PROGRAM Y_Master_Y_Axis
VAR
	
	// Link to Task
	refY_Axis							:AXIS_REF;	//Axis_1
										
										
	fPositionLimitMin					:LREAL			 := 5;
	fPositionLimitMax					:LREAL			 := 110;
	fLimitPositionLow					:LREAL; 		//16#0001_000D
	fLimitPositionHigh					:LREAL;			//16#0001_000E
	
	// Local Axis Config
	posTarget							:LREAL;
	fOffsets							:ARRAY [1..3]OF LREAL;
	nOfSetPos							:INT:=3;
	fCurrentPosition					:LREAL;

    // State Machine CTRL
    eState								:E_AxisState:=E_AxisState.ABORTED;

	// Timers && Triggers
	tonResetError						:Tc2_Standard.TON;
	tonPowerAxis						:Tc2_Standard.TON;
	tonPowerAxis2						:Tc2_Standard.TON;
	tonActionDone						:Tc2_Standard.TON;
	tonMoveTimeout						:Tc2_Standard.TON;
	tonPowerUpTimeout					:Tc2_Standard.TON;
	tonPowerUpError						:Tc2_Standard.TON;
	tonAbortModule						:Tc2_Standard.TON;
	tonDelayExe							:Tc2_Standard.TON;

				
    // Motion FB Instances
    fbPower    							:Tc2_MC2.MC_Power;
    fbReset    							:Tc2_MC2.MC_Reset;
    fbStop     							:Tc2_MC2.MC_Stop;
    fbMoveABS     						:Tc2_MC2.MC_MoveAbsolute;
	fbMoveREL							:Tc2_MC2.MC_MoveRelative;
	fbReadStatus						:Tc2_MC2.MC_ReadStatus;
	fbReadPos							:Tc2_MC2.MC_ReadActualPosition;
	stAxisStatus						:ST_AxisStatus;
	fbParameter							:ARRAY[0..1]OF Tc2_MC2.MC_ReadParameter;
	
	// Function Blocks Flags
	bReq_Power							:BOOL;		// Request Power to Axis 
	bReq_Reset							:BOOL;		// Request Axis Reset
	bReq_MoveABS						:BOOL;		// Request Move Action 
	bReq_MoveREL						:BOOL;		// Request Move Action
	bReq_Stop							:BOOL;		// Request Axis to Stop
	bAxisInError						:BOOL;
	
	//Index
	idx									:INT;
	//MANUAL MODE
	nManualModeState					:DINT;
	trigbMoveToPos						:R_TRIG;
	bTest								:BOOL;

//-------------------------------------------------------------------------------*		
END_VAR
VAR_INPUT	
	bRetract							:BOOL;		// Velocity Change
END_VAR
VAR PERSISTENT
		// Set Parameters
    cfgAxis    							:ST_Y_Axis;(*:=(
										posHome 		  := 7.0,
										posWorkPositions := [14.5,33.7,100.0],
										fPositionOffsets := [0.0,  0.0,  0.0],
										fTargetVelocity  := 25.0,
										fRetractVelocity := 90.0);//after comes from hmi*)
END_VAR

//--------------------IN/OUT-----------------------------------------------------*
VAR_INPUT	
	CMD									:ST_ModuleCMD;	
END_VAR
VAR_OUTPUT	
	STATUS								:ST_ModuleStatus;	
END_VAR
//------------------------------------------------------------------------oldschoo1

PRG_Fault_Axis_Y(aAlarms := GVL_Master.stAlarms);
// Positions Offsets Mapping
IF (GVL_PERSISTENT.fPositions_Offset[1]>1.3) OR (GVL_PERSISTENT.fPositions_Offset[2]>1.3)
	THEN
fOffsets[1] := 0.0;
fOffsets[2] := 0.0;
ELSE
fOffsets[1] := GVL_PERSISTENT.fPositions_Offset[1];	//Picking Screw Position
fOffsets[2] := GVL_PERSISTENT.fPositions_Offset[2];	//Screwwing and Pressing Actions Position	
END_IF

//-------------------------------------------------------------------------------------------*
//Call For Actions
a_Ctrl_Axis();
b_Call_AxisFBs();
d_Get_CurrentPosition();
//---------------------*
//------------------------------------------------------------------------------------oldschoo1

ACTION a_Ctrl_Axis:
// Timmers && Triggers     
tonPowerAxis	(IN:= eState=E_AxisState.ENABLE_POWER, 
			 	 PT:= T#50MS);			 
tonActionDone	(IN:= eState=E_AxisState.IN_TARGET_POS,
			  	 PT:= T#100MS);
tonMoveTimeout	(IN:= eState=E_AxisState.MOVE_ABS OR eState=E_AxisState.MOVE_REL,
			   	 PT:= T#10S);			  
tonAbortModule	(IN:=	cmd.bAbort OR (NOT stSafety.bSafety_OK) OR (NOT cmd.bEnable),
			     PT:= T#100MS);
tonResetError	(IN:= cmd.bReset OR fbPower.Error OR fbStop.Error OR fbMoveABS.Error OR fbMoveREL.Error,
			  	 PT:= T#500MS);
tonDelayExe  	(IN:= eState=E_AxisState.HOMING AND stY_Axis.bSetToHome,
			  	 PT:= T#300MS);
(**************************************************RESET************************************************)		   
// Reset Errors
IF cmd.bReset OR fbPower.Error OR fbStop.Error OR fbMoveABS.Error OR fbMoveREL.Error THEN

			status.bError 	:= TRUE;
			bReq_Power 		:= FALSE;
			bReq_MoveABS 	:= FALSE;
			bReq_MoveREL 	:= FALSE;
			bReq_Stop 		:= FALSE;		
            eState := E_AxisState.RESET_ERROR;
			END_IF
IF  eState=E_AxisState.ABORTED THEN
CMD_Axis.bExecute			  :=FALSE;
stY_Axis.bSetToHome			  :=FALSE;
Y_Master_Y_Axis.bRetract 	  :=FALSE; END_IF			
IF tonResetError.Q THEN bReq_Reset := TRUE; END_IF
IF bAxisInError THEN bReq_Reset:=bResetButtonRisingEdge; eState:= E_AxisState.ERROR; END_IF

// Abort Action
IF tonAbortModule.Q THEN

			bReq_Power := FALSE;
			eState := E_AxisState.ABORTED;
			END_IF
IF CMD.bManualMode THEN
	eState := E_AxisState.MANUAL_MODE;
END_IF
(*******************************************************CTRL***********************************************************)
// Axis CTRL State Machine
CASE eState OF //--------------------------------------------------------------------------------------------------SM
	
E_AxisState.ABORTED://-------------------------------------------------------------------------------------------ABORTED:


							IF stSafety.bSafety_OK AND cmd.bEnable AND NOT fbPower.Error THEN
								
									bReq_Power := TRUE;
									eState := E_AxisState.ENABLE_POWER;
							END_IF

E_AxisState.ENABLE_POWER://---------------------------------------------------------------------------------ENABLE_POWER:

							IF fbPower.Status AND NOT fbPower.Error THEN
								
									bReq_Reset := TRUE;
									eState := E_AxisState.HOMING;
							END_IF

E_AxisState.RESET_ERROR://-----------------------------------------------------------------------------------RESET_ERROR:

							IF fbReset.Done AND fbPower.Status THEN
								
									bReq_Reset := FALSE;
									eState := E_AxisState.HOMING;
									
							ELSIF fbReset.Done AND NOT fbPower.Status THEN
							
										eState := E_AxisState.ABORTED;
										
							ELSIF NOT fbPower.Error AND NOT fbStop.Error AND 
								  NOT fbMoveABS.Error AND NOT fbMoveREL.Error THEN
								  
										eState := E_AxisState.ABORTED;
							END_IF

E_AxisState.HOMING://---------------------------------------------------------------------------------------------HOMING:

							IF ABS(fCurrentPosition - cfgAxis.posHome)<=0.5 THEN
								
										bReq_MoveABS				  :=FALSE;
										CMD_Axis.bExecute			  :=FALSE;
										stY_Axis.bSetToHome			  :=FALSE;
										Y_Master_Y_Axis.bRetract 	  :=FALSE;
										
										eState := E_AxisState.AXIS_READY;	
 							ELSE
										//bReq_MoveABS				  :=TRUE; //test
										stY_Axis.bSetToHome			  :=TRUE;
										posTarget:=cfgAxis.posHome;
										Y_Master_Y_Axis.bRetract 	  :=TRUE;
										eState 							:= E_AxisState.MOVE_ABS;
							END_IF
							 	
									IF tonDelayExe.Q THEN
											CMD_Axis.bExecute		  :=TRUE;
									END_IF
									
E_AxisState.AXIS_READY://-------------------------------------------------------------------------------------AXIS_READY:

							IF cmd.bExecute THEN
									eState := E_AxisState.GET_TARGET;
							END_IF
							
E_AxisState.GET_TARGET://-------------------------------------------------------------------------------------GET_TARGET:

							posTarget := c_Get_TargetPositon(
															posHome 	:= cfgAxis.posHome,
															posPoints   := cfgAxis.posWorkPositions,
															fOffsets	:= fOffsets,
															bSetHome 	:= stY_Axis.bSetToHome,
															bSetPoint 	:= stY_Axis.bSetToPosition
															);	
															eState := E_AxisState.MOVE_ABS;
	
E_AxisState.MOVE_ABS://-----------------------------------------------------------------------------------------MOVE_ABS:

							IF posTarget > fPositionLimitMin AND
							   posTarget < fPositionLimitMax
 								THEN 
									bReq_MoveABS := TRUE;
									eState := E_AxisState.MOVING_ABS;
							END_IF
							stY_Axis.bSetToHome			  :=FALSE;
							
							
E_AxisState.MOVING_ABS://-------------------------------------------------------------------------------------MOVING_ABS:

							IF fbMoveABS.Done THEN
									
									bReq_MoveABS := FALSE;
									eState := E_AxisState.IN_TARGET_POS;
									
							ELSIF tonMoveTimeout.Q THEN
									
									bReq_MoveABS := FALSE;
									eState := E_AxisState.ERROR;
							END_IF
							//TO KNOW POSITION OF AXIS
							GVL_HMI.bY_AxisInPosition1		:= FALSE;
							GVL_HMI.bY_AxisInPosition2		:= FALSE;
							GVL_HMI.bY_AxisInPosition3		:= FALSE;
							GVL_HMI.bY_AxisInHomePosition	:= FALSE;

E_AxisState.MOVE_REL:;
E_AxisState.MOVING_REL:;

E_AxisState.IN_TARGET_POS://-------------------------------------------------------------------------------IN_TARGET_POS:

							IF tonActionDone.Q THEN
								eState := E_AxisState.AXIS_READY;
							END_IF
							//TO KNOW THE POSITION OF THE AXIS
							IF stY_Axis.bSetToPosition[1] THEN
								GVL_HMI.bY_AxisInPosition1				:= TRUE;
							END_IF
							IF stY_Axis.bSetToPosition[2] THEN
								GVL_HMI.bY_AxisInPosition2				:= TRUE;
							END_IF
							IF stY_Axis.bSetToPosition[3] THEN
								GVL_HMI.bY_AxisInPosition3				:= TRUE;
							END_IF
							IF stY_Axis.bSetToHome THEN
								GVL_HMI.bY_AxisInHomePosition			:= TRUE;
							END_IF
E_AxisState.ERROR://-----------------------------------------------------------------------------------------------ERROR:

	 					eState := E_AxisState.ABORTED;
						
E_AxisState.MANUAL_MODE://-----------------------------------------------------------------------------------MANUAL_MODE:

							e_Manual();
					
							IF NOT CMD.bManualMode THEN
								eState := E_AxisState.ABORTED;
							END_IF

ELSE 
eState := E_AxisState.ABORTED;
END_CASE //------------------------------------------------------------------------------------------------------END_CASE

(******************************************************STATUS************************************************************)
// Module Status
status.bReady	:= eState = E_AxisState.AXIS_READY;

status.bBusy	:= eState <> E_AxisState.ABORTED	AND
				   eState <> E_AxisState.AXIS_READY AND
				   eState <> E_AxisState.IN_TARGET_POS AND
				   eState <> E_AxisState.ERROR;
				   
status.bDone	:= eState = E_AxisState.IN_TARGET_POS;

status.bError	:= eState = E_AxisState.ERROR OR 
				   fbPower.Error OR fbStop.Error OR fbMoveABS.Error OR fbMoveREL.Error; 
//---------------------------------------------------------------------------------------------------------------oldschoo1
END_ACTION

ACTION b_Call_AxisFBs:
// CTRL FBs Call

	fbPower 	(Axis:=refY_Axis, Enable:=bReq_Power, Enable_Positive:=bReq_Power, Enable_Negative:=bReq_Power);
	fbReset 	(Axis:=refY_Axis, Execute:=bReq_Reset);
	
  fbMoveABS 	(Axis:=refY_Axis, Execute:=bReq_MoveABS, 
				 Position:=posTarget, Velocity:= SEL(bRetract,cfgAxis.fTargetVelocity,cfgAxis.fRetractVelocity));
  fbMoveREL 	(Axis:=refY_Axis, Execute:=FALSE);
 	 fbStop 	(Axis:=refY_Axis, Execute:=FALSE);
  fbReadPos		(Axis:=refY_Axis, Enable:=eState=E_AxisState.HOMING);
fbParameter[0]  (Axis:=refY_Axis, Enable:=TRUE, ParameterNumber:=MC_AXISPARAMETER.AxisMinSoftPosLimit, Value=>fLimitPositionLow);
fbParameter[1]  (Axis:=refY_Axis, Enable:=TRUE, ParameterNumber:=MC_AXISPARAMETER.AxisMaxSoftPosLimit, Value=>fLimitPositionHigh);
fbReadStatus	(Axis:=refY_Axis, Enable:=TRUE, Status=>stAxisStatus, Error=>bAxisInError);
//-----------------------------------------------------------------------------------------------------------------------oldschoo1
END_ACTION

METHOD c_Get_TargetPositon	:LREAL
VAR_INPUT

	// Positions
    posHome     			:LREAL;
    posPoints   			:ARRAY[1..3]OF LREAL;
    fOffsets  				:ARRAY[1..3]OF LREAL;
	
	// Set Target Flags
    bSetHome    			:BOOL;
    bSetPoint   			:ARRAY[1..3]OF BOOL;
	
END_VAR
//----------------------------------------------------------oldschoo1


VAR
	idx           			:INT;
	posTargeteBase	     	:LREAL;
END_VAR
IF bSetHome THEN
    		posTargeteBase := posHome;
ELSE
	
			FOR idx:= 1 TO 3 
			DO
					IF bSetPoint[idx] THEN
						posTargeteBase := posPoints[idx] + fOffsets[idx];
						EXIT;
					END_IF		
			END_FOR
END_IF

c_Get_TargetPositon	:= posTargeteBase;
//--------------------------------------------------------------oldschoo1
END_METHOD

ACTION d_Get_CurrentPosition:
IF fbReadPos.Valid THEN fCurrentPosition:=fbReadPos.Position; END_IF
//----------------------------------------------------------oldschoo1
END_ACTION

ACTION e_Manual:
posTarget := c_Get_TargetPositon(
															posHome 	:= cfgAxis.posHome,
															posPoints   := cfgAxis.posWorkPositions,
															fOffsets	:= fOffsets,
															bSetHome 	:= stY_Axis.bSetToHome,
															bSetPoint 	:= stY_Axis.bSetToPosition
															);	
trigbMoveToPos( CLK := GVL_HMI.bMoveToPos );
IF GVL_HMI.bY_AxisPosition1 THEN
	stY_Axis.bSetToPosition[1]			:= TRUE;
	GVL_HMI.bMoveToPos					:= TRUE;
END_IF
IF GVL_HMI.bY_AxisPosition2 THEN
	stY_Axis.bSetToPosition[2]			:= TRUE;
	GVL_HMI.bMoveToPos					:= TRUE;
END_IF
IF GVL_HMI.bY_AxisPosition3 THEN
	stY_Axis.bSetToPosition[3]			:= TRUE;
	GVL_HMI.bMoveToPos					:= TRUE;
END_IF
IF GVL_HMI.bY_HomePosition THEN
	stY_Axis.bSetToHome					:= TRUE;
	GVL_HMI.bMoveToPos					:= TRUE;
END_IF
	
IF trigbMoveToPos.Q THEN
	nManualModeState					:=10;
END_IF

CASE nManualModeState OF
	
10:
IF posTarget > fPositionLimitMin AND
		posTarget < fPositionLimitMax THEN 
		bReq_MoveABS 					:= TRUE;
		GVL_HMI.bY_AxisInPosition1Man	:= FALSE;
		GVL_HMI.bY_AxisInPosition2Man	:= FALSE;
		GVL_HMI.bY_AxisInPosition3Man	:= FALSE;
		GVL_HMI.bY_AxisInHomePositionMan:= FALSE;
		nManualModeState				:=20;
	END_IF	
20:
IF fbMoveABS.Done THEN	
	IF stY_Axis.bSetToPosition[1] THEN
		GVL_HMI.bY_AxisInPosition1Man	:= TRUE;
	END_IF
	IF stY_Axis.bSetToPosition[2] THEN
		GVL_HMI.bY_AxisInPosition2Man	:= TRUE;
	END_IF
	IF stY_Axis.bSetToPosition[3] THEN
		GVL_HMI.bY_AxisInPosition3Man	:= TRUE;
	END_IF
	IF stY_Axis.bSetToHome THEN
		GVL_HMI.bY_AxisInHomePositionMan:= TRUE;
	END_IF
	nManualModeState					:=30;
END_IF
	
30:								
		bReq_MoveABS 					:= FALSE;
		stY_Axis.bSetToPosition[1]		:= FALSE;
		stY_Axis.bSetToPosition[2]		:= FALSE;
		stY_Axis.bSetToPosition[3]		:= FALSE;
		stY_Axis.bSetToHome				:= FALSE;
		GVL_HMI.bMoveToPos				:= FALSE;
		
IF NOT GVL_Master.stMachineStatus.bManualMode THEN
		GVL_HMI.bY_AxisInPosition1Man	:= FALSE;
		GVL_HMI.bY_AxisInPosition2Man	:= FALSE;
		GVL_HMI.bY_AxisInPosition3Man	:= FALSE;
		GVL_HMI.bY_AxisInHomePositionMan:= FALSE;
END_IF
END_CASE
END_ACTION

END_PROGRAM

(* stored: Version 1.1.0.1, ProductVersion 3.1.4024.12
   POU Y_Master_Y_Axis: Id {d3204fea-0ebc-46da-b5e6-c7a8a4e9a82e}, SpecialFunc None
   Action a_Ctrl_Axis: Id {4981aca3-a94a-4db5-9a82-6e46587d07a9}
   Action b_Call_AxisFBs: Id {46e77f9d-ddc0-4859-9573-a3495da6c21a}
   Method c_Get_TargetPositon: Id {d69107da-47c7-40a8-b230-3defd16f8c05}
   Action d_Get_CurrentPosition: Id {799ecc77-506d-4eda-a5b2-07b88c5b9039}
   Action e_Manual: Id {626d8992-b5ab-4015-adbc-a66765231fb7} *)
